// TIA Portal V17 export
// export: Created 2022-07-05T08:49:25.2952625Z, ExportSetting WithDefaults, DisplayName Totally Integrated Automation Portal, DisplayVersion V17, DisplayName TIA Portal Openness, DisplayVersion V17, DisplayName TIA Portal Version Control Interface, DisplayVersion V17, DisplayName STEP 7 Professional, DisplayVersion V17, DisplayName STEP 7 Safety, DisplayVersion V17, DisplayName WinCC Advanced, DisplayVersion V17
DATA_BLOCK "InstOPCMethodSetMachineTime"   // DB3
VERSION : 0.1
// stored: AutoNumber true, DBAccessibleFromOPCUA true, DBAccessibleFromWebserver true, InstanceOfName OPCMethodSetMachineTime, InstanceOfType FB
"OPCMethodSetMachineTime"
   // VAR
   //    OPC_UA_ServerMethodPre_Instance { S7_SetPoint := 'True'} : OPC_UA_ServerMethodPre;
   //    statUAMStatusPre { S7_SetPoint := 'True'} : "typeOPCUAStatus";
   //    statUAMStatusPost { S7_SetPoint := 'True'} : "typeOPCUAStatus";
   //    UAMethod_InParameters : Struct
   //       DateTime : LDT;
   //    END_STRUCT;
   //    OPC_UA_ServerMethodPost_Instance { S7_SetPoint := 'True'} : OPC_UA_ServerMethodPost;
   // END_VAR
BEGIN
END_DATA_BLOCK
